INTERFACE I_MotionInterlocks

PROPERTY AllBackwardEnabled : BOOL
GET
END_GET
END_PROPERTY

PROPERTY AllEnabled : BOOL
GET
END_GET
END_PROPERTY

PROPERTY AllForwardEnabled : BOOL
GET
END_GET
END_PROPERTY

PROPERTY EPSBackwardEnable : BOOL
GET
END_GET
SET
END_SET
END_PROPERTY

PROPERTY EPSForwardEnable : BOOL
GET
END_GET
SET
END_SET
END_PROPERTY

PROPERTY EPSPowerEnable : BOOL
GET
END_GET
SET
END_SET
END_PROPERTY

PROPERTY Error : BOOL
GET
END_GET
END_PROPERTY

PROPERTY ErrorID : UDINT
GET
END_GET
END_PROPERTY

PROPERTY GantryAxis : BOOL
GET
END_GET
SET
END_SET
END_PROPERTY

PROPERTY GantryBackwardEnable : BOOL
GET
END_GET
SET
END_SET
END_PROPERTY

PROPERTY GantryForwardEnable : BOOL
GET
END_GET
SET
END_SET
END_PROPERTY

PROPERTY HardwareEnable : BOOL
GET
END_GET
SET
END_SET
END_PROPERTY

PROPERTY InterlockOk : BOOL
GET
END_GET
END_PROPERTY

PROPERTY LimBwdEnable : BOOL
GET
END_GET
SET
END_SET
END_PROPERTY

PROPERTY LimFwdEnable : BOOL
GET
END_GET
SET
END_SET
END_PROPERTY

PROPERTY LimHit : BOOL
GET
END_GET
END_PROPERTY

PROPERTY LimHitIdling : BOOL
GET
END_GET
END_PROPERTY

PROPERTY LimHitMoving : BOOL
GET
END_GET
END_PROPERTY

PROPERTY LimHome : BOOL
GET
END_GET
SET
END_SET
END_PROPERTY

PROPERTY PowerSelf : BOOL
GET
END_GET
SET
END_SET
END_PROPERTY

PROPERTY SafetyReady : BOOL
GET
END_GET
END_PROPERTY

PROPERTY SoftInterlock : BOOL
GET
END_GET
SET
END_SET
END_PROPERTY

PROPERTY UserEnable : BOOL
GET
END_GET
END_PROPERTY

PROPERTY WarnID : UINT
GET
END_GET
END_PROPERTY

PROPERTY WarningMsg : STRING
GET
END_GET
END_PROPERTY

END_INTERFACE

(* stored: Version 1.1.0.1
   Itf I_MotionInterlocks: Id {7ac89254-d732-4980-b014-871a72f21fa7}
   Property AllBackwardEnabled: Id {44fa7548-c01f-4da3-a333-2275934d3112}
   Get Get: Id {8e243d13-164d-4d5d-8112-387f3a8b0fca}
   Property AllEnabled: Id {4d69c415-64ae-45e5-8741-9ee750fa41cf}
   Get Get: Id {09b8b64d-72b0-467d-b693-fa3e229ceb18}
   Property AllForwardEnabled: Id {3ce5ac2e-1c09-4fd1-941c-2cbe06026596}
   Get Get: Id {8ac731aa-4431-4ad2-aad0-76448e67d881}
   Property EPSBackwardEnable: Id {9b6fa1bd-6512-4d3d-85db-8498ddd7669c}
   Get Get: Id {e34fca84-01bf-4e87-aa6d-c77abdad8429}
   Set Set: Id {4ec5e289-3899-4d94-b3b7-ea5f59d60aff}
   Property EPSForwardEnable: Id {ae0d8c46-3803-4d4d-bfc2-e4e8d9e9b7f4}
   Get Get: Id {4c46cb3f-211f-4da9-a32e-77acf2d34ed0}
   Set Set: Id {0a7eaec5-5dc1-4ab5-bd95-124bb3e3ced6}
   Property EPSPowerEnable: Id {2ab43de3-0abf-4f29-b1d9-776886efae5d}
   Get Get: Id {963baa30-2ed7-4807-8ba8-e09808456204}
   Set Set: Id {8bc5bd75-07a7-44de-ac8f-1ad8ff551029}
   Property Error: Id {e7bf6778-c6b9-4c5a-b105-4d2a2c94dadc}
   Get Get: Id {e4d10e81-4cda-4fea-b6c9-9cbe365e367c}
   Property ErrorID: Id {052a5e61-bd0b-473b-8c73-0685a48edd45}
   Get Get: Id {f9a6101a-75a4-46b6-a241-3924343635ff}
   Property GantryAxis: Id {56006ae1-c693-47b5-a7b2-3327681468a5}
   Get Get: Id {29ac787b-548b-40c0-aee0-72e462d082cc}
   Set Set: Id {46c657f3-a086-4fed-b359-12c3fd9d60d1}
   Property GantryBackwardEnable: Id {f904ecbf-7926-4b97-a553-c1e262839afe}
   Get Get: Id {f53ef5a8-39bd-4b60-8938-d7e59932b51a}
   Set Set: Id {a5df2c27-bd1f-4e41-b211-426d9f0beb2c}
   Property GantryForwardEnable: Id {a1dbb698-133c-46e9-819b-17b9b9f21b23}
   Get Get: Id {bd086b46-a9ef-4695-a19b-7f1e76359447}
   Set Set: Id {35f02b45-8b53-4e6a-9812-d446b45c27b1}
   Property HardwareEnable: Id {855c6e4b-bfed-49b3-bdec-eafa65093aa9}
   Get Get: Id {3bc8c738-8360-4ae7-9ad5-cf8bc24dacf1}
   Set Set: Id {489a79c4-eb9c-4a2f-baad-54d7878ac34a}
   Property InterlockOk: Id {1f6b357a-4433-42e5-8fa2-bf574bca239f}
   Get Get: Id {9855daed-54fd-4c0d-8687-1dc62a376c17}
   Property LimBwdEnable: Id {4f071531-664b-43fb-9b98-46ce706701d6}
   Get Get: Id {9187b4a7-a42c-4364-a237-fe27d1b092b0}
   Set Set: Id {b9aff11f-e55e-4ea0-a544-b45c3be44f95}
   Property LimFwdEnable: Id {63378470-96d4-47b7-a381-4d50609bb5a2}
   Get Get: Id {13bb15a4-f20a-4eed-b421-340a7c7204a2}
   Set Set: Id {7ad36303-dc71-4d7a-b996-eaec00eed2df}
   Property LimHit: Id {00f31b83-20b0-4e18-bb57-b84a58adcd1b}
   Get Get: Id {dc48a399-6ef3-4f49-9589-4858181b8029}
   Property LimHitIdling: Id {a9898372-986c-4ee4-bc98-43640fd003f2}
   Get Get: Id {d9233391-3505-4407-ade5-ca790ab05516}
   Property LimHitMoving: Id {12768a8b-8e2d-462d-ac59-05ed276cdf42}
   Get Get: Id {f40fa498-6562-48ff-8455-7f34f6bbcf01}
   Property LimHome: Id {43b3c4e0-2529-4ca2-94b6-01308791bd0f}
   Get Get: Id {fa4d37b3-5d02-4b73-968e-4a37c39a113f}
   Set Set: Id {aca26340-7624-4f3a-8bc3-b354a8230aaf}
   Property PowerSelf: Id {af7539d4-48fa-4915-a716-1585614bb150}
   Get Get: Id {832ea85a-44e1-43f2-84fb-a9a7ce8a9a54}
   Set Set: Id {3ab08d4c-6e93-4a5c-b644-d0f7e3500942}
   Property SafetyReady: Id {c4a49c88-eac4-4e17-84d8-41063fa69887}
   Get Get: Id {67ae7808-2d1e-4903-92a5-9e496ca319df}
   Property SoftInterlock: Id {84b462fb-97b6-4df9-b44c-e4fc3600b4a1}
   Get Get: Id {4c848c4c-616c-4dea-8b19-c0ad93f2399c}
   Set Set: Id {7e455863-b97d-4ef2-8c0a-175169e8ec44}
   Property UserEnable: Id {b04015ea-94bc-4cb0-a1f4-ebb6556cce84}
   Get Get: Id {3936eba9-09b5-408d-b793-738e943f6fd9}
   Property WarnID: Id {be859d4c-20b0-48fc-90e8-64961601a870}
   Get Get: Id {aff35a25-4efa-4678-8127-c8619732e505}
   Property WarningMsg: Id {bf7b81d5-c154-46fb-b50d-9188e5c9721a}
   Get Get: Id {904bcd85-b16b-4196-9319-f47b5feeb0d9} *)
